Omron Sysmac Studio project Proyecto_1 (Sysmac Studio 1.23.0.14, StandardProject)

# Controller new_Controller_0: NX1P2-1040DT1 version 1.18
Task PrimaryTask (priority 4, period or condition 2000): Programa0

VAR_GLOBAL
    PM : BOOL;  (* Pulsador de Marcha; at BuiltInIO://cpu/#0/Input_Bit_00 *)
    PP : BOOL;  (* Pulsador de Parada; at BuiltInIO://cpu/#0/Input_Bit_01 *)
    S1 : BOOL;  (* Final de Carrera 1; at BuiltInIO://cpu/#0/Input_Bit_02 *)
    S2 : BOOL;  (* Final de Carrera 2; at BuiltInIO://cpu/#0/Input_Bit_03 *)
    KM1 : BOOL;  (* Contactor Marcha Izquierda; at BuiltInIO://cpu/#0/Output_Bit_00 *)
    KM2 : BOOL;  (* Contactor Marcha Derecha; at BuiltInIO://cpu/#0/Output_Bit_01 *)
END_VAR

PROGRAM Programa0
VAR
    Et0 : BOOL;  (* Etapa 0 *)
    Et1 : BOOL;  (* Etapa 1 *)
    Et2 : BOOL;  (* Etapa 2 *)
    T1 : TON;
    T2 : TON;
END_VAR
VAR_EXTERNAL
    S2 : BOOL;
    PM : BOOL;
    PP : BOOL;
    S1 : BOOL;
    KM1 : BOOL;
    KM2 : BOOL;
END_VAR

(* Section Secuencial: ladder, written here as Structured Text *)

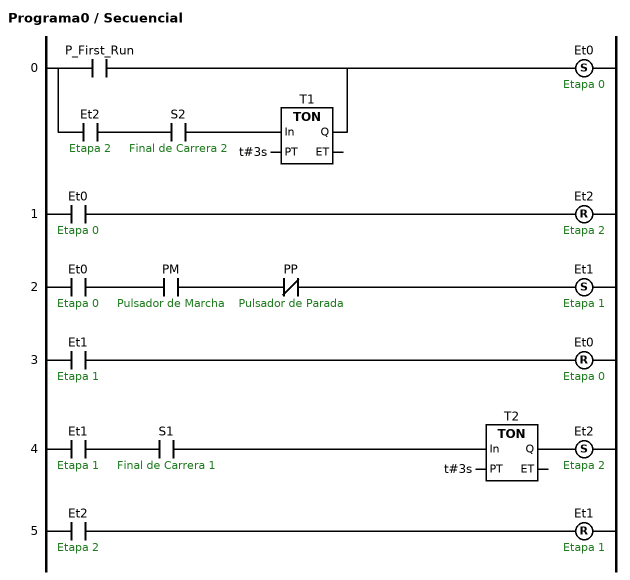
(* Rung 0 *)
T1(In := Et2 AND S2, PT := t#3s);
IF P_First_Run OR T1.Q THEN Et0 := TRUE; END_IF;
(* Rung 1 *)
IF Et0 THEN Et2 := FALSE; END_IF;
(* Rung 2 *)
IF Et0 AND PM AND NOT PP THEN Et1 := TRUE; END_IF;
(* Rung 3 *)
IF Et1 THEN Et0 := FALSE; END_IF;
(* Rung 4 *)
T2(In := Et1 AND S1, PT := t#3s);
IF T2.Q THEN Et2 := TRUE; END_IF;
(* Rung 5 *)
IF Et2 THEN Et1 := FALSE; END_IF;

(* Section Salidas: ladder, written here as Structured Text *)

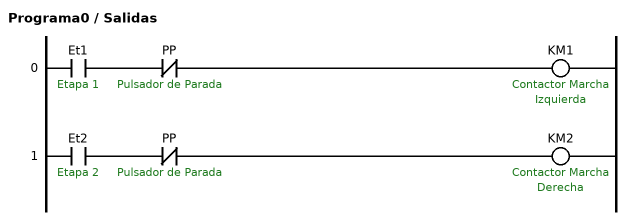
(* Rung 0 *)
KM1 := Et1 AND NOT PP;
(* Rung 1 *)
KM2 := Et2 AND NOT PP;
END_PROGRAM